// TIA Portal V17 export
// export: Created 2024-08-26T21:10:53.4753687Z, ExportSetting WithDefaults, DisplayName Totally Integrated Automation Portal, DisplayVersion V17 Update 7, DisplayName TIA Portal Openness, DisplayVersion V17 Update 7, DisplayName TIA Portal Version Control Interface, DisplayVersion V17, DisplayName SINAMICS Startdrive Advanced, DisplayVersion V17 SP2, DisplayName SINAMICS Startdrive G110M, G120, G120C, G120D, G120P, G115D, DisplayVersion V17 SP2, DisplayName SINAMICS Startdrive G130, G150, S120, S150, SINAMICS MV, S210, DisplayVersion V17 SP2, DisplayName STEP 7 Professional, DisplayVersion V17 Update 7, DisplayName STEP 7 Safety, DisplayVersion V17 Update 6, DisplayName WinCC Advanced / Unified PC, DisplayVersion V17 Update 7
VAR_GLOBAL   // PLC tag table "powerFocus6000"
   counterClockwiseDirection AT %I182.5 : Bool;
   clockwiseDirection AT %I182.6 : Bool;
   torqueOk AT %I19.6 : Bool;
   torqueDone AT %I20.0 : Bool;
   torqueNok AT %I19.7 : Bool;
   finalTorqueInt1 AT %IW13 : Word;
   finalTorqueDecimal1 AT %IW15 : Word;
   deactivateTool AT %Q17.7 : Bool;
   activateTorqueTool AT %Q17.0 : Bool;
   clearNestScanerRead AT %Q4.0 : Bool;
   torqueInputSelect AT %QB18 : Byte;
   thighteningStart AT %Q17.3 : Bool;
   correctTorque AT %M3.5 : Bool;
   p6000Test1 AT %M152.1 : Bool;
   p6000Test2 AT %M152.2 : Bool;
   p6000Test3 AT %M152.3 : Bool;
   p6000Test1Enabled AT %M152.4 : Bool;
   p6000Test2Enabled AT %M152.5 : Bool;
   p6000Test3Enabled AT %M152.6 : Bool;
   counterClockwiseDirectionWarning AT %M23.0 : Bool;
   clockwiseDirectionWarning AT %M23.1 : Bool;
   hmiFinalTorqueDecimal AT %MW214 : Word;
   hmiFinalTorqueInt AT %MW212 : Word;
END_VAR
